// LS Electric XG5000 project: Packing_Machine_NEW1
// PLC NewPLC
// module base 0 slot 0: Input/Output Module:XBC-DN/DP32U (DC 24V Input 16 Contacts, Transistor Output 16 Contacts)
// module base 0 slot 1: Internal Positioning:XBF-PD04E (Position Control  Pulse(LD), Output Type(4 axis))

PROGRAM Program (task: Scan Program)

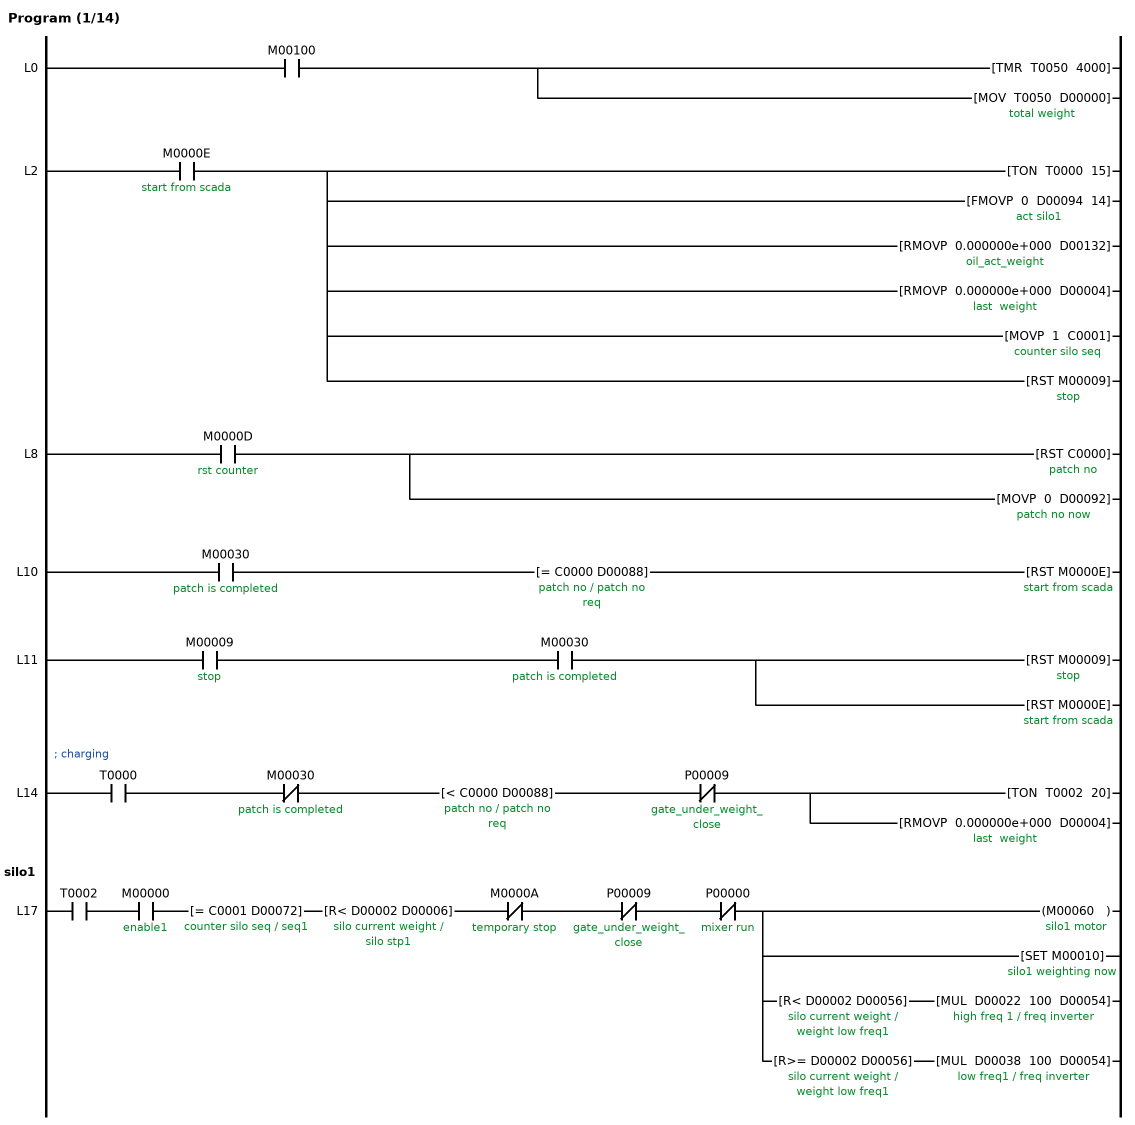
; L0
LOAD      M00100
TMR       T0050 4000
MOV       T0050 D00000	// total weight
; L2
LOAD      M0000E	// start from scada
TON       T0000 15
FMOVP     0 D00094 14	// act silo1
RMOVP     0.000000e+000 D00132	// oil_act_weight
RMOVP     0.000000e+000 D00004	// last  weight
MOVP      1 C0001	// counter silo seq
RST       M00009	// stop
; L8
LOAD      M0000D	// rst counter
RST       C0000	// patch no
MOVP      0 D00092	// patch no now
; L10
LOAD      M00030	// patch is completed
AND=      C0000 D00088	// patch no / patch no req
RST       M0000E	// start from scada
; L11
LOAD      M00009	// stop
AND       M00030	// patch is completed
RST       M00009	// stop
RST       M0000E	// start from scada
// charging
; L14
LOAD      T0000
AND NOT   M00030	// patch is completed
AND<      C0000 D00088	// patch no / patch no req
AND NOT   P00009	// gate_under_weight_close
TON       T0002 20
RMOVP     0.000000e+000 D00004	// last  weight
silo1:
; L17
LOAD      T0002
AND       M00000	// enable1
AND=      C0001 D00072	// counter silo seq / seq1
ANDR<     D00002 D00006	// silo current weight / silo stp1
AND NOT   M0000A	// temporary stop
AND NOT   P00009	// gate_under_weight_close
AND NOT   P00000	// mixer run
OUT       M00060	// silo1 motor
SET       M00010	// silo1 weighting now
MPUSH
ANDR<     D00002 D00056	// silo current weight / weight low freq1
MUL       D00022 100 D00054	// high freq 1 / freq inverter
MPOP
ANDR>=    D00002 D00056	// silo current weight / weight low freq1
MUL       D00038 100 D00054	// low freq1 / freq inverter

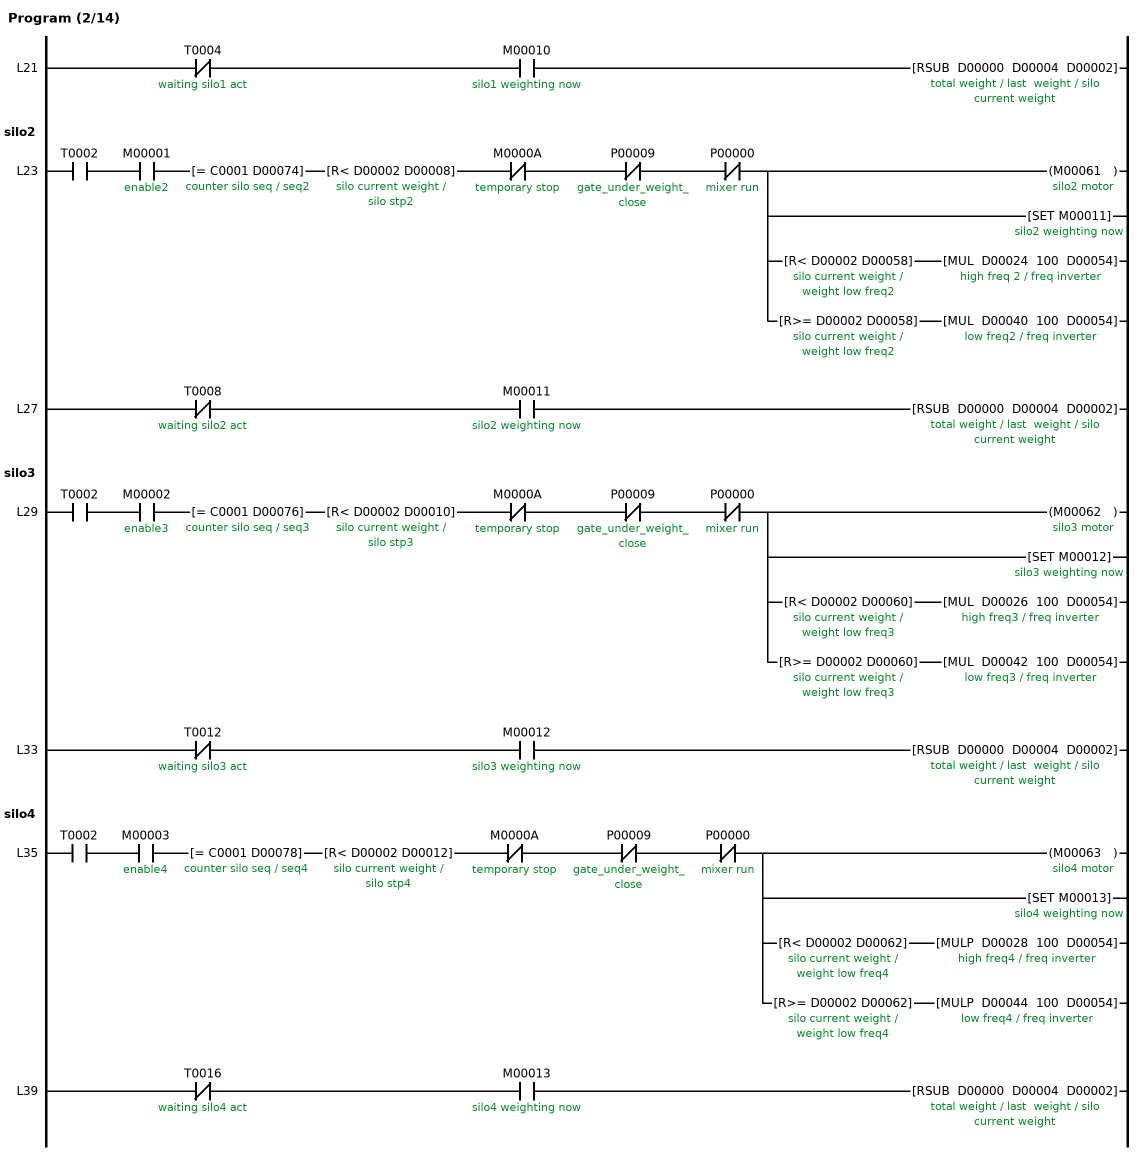
; L21
LOAD NOT  T0004	// waiting silo1 act
AND       M00010	// silo1 weighting now
RSUB      D00000 D00004 D00002	// total weight / last  weight / silo current weight
silo2:
; L23
LOAD      T0002
AND       M00001	// enable2
AND=      C0001 D00074	// counter silo seq / seq2
ANDR<     D00002 D00008	// silo current weight / silo stp2
AND NOT   M0000A	// temporary stop
AND NOT   P00009	// gate_under_weight_close
AND NOT   P00000	// mixer run
OUT       M00061	// silo2 motor
SET       M00011	// silo2 weighting now
MPUSH
ANDR<     D00002 D00058	// silo current weight / weight low freq2
MUL       D00024 100 D00054	// high freq 2 / freq inverter
MPOP
ANDR>=    D00002 D00058	// silo current weight / weight low freq2
MUL       D00040 100 D00054	// low freq2 / freq inverter
; L27
LOAD NOT  T0008	// waiting silo2 act
AND       M00011	// silo2 weighting now
RSUB      D00000 D00004 D00002	// total weight / last  weight / silo current weight
silo3:
; L29
LOAD      T0002
AND       M00002	// enable3
AND=      C0001 D00076	// counter silo seq / seq3
ANDR<     D00002 D00010	// silo current weight / silo stp3
AND NOT   M0000A	// temporary stop
AND NOT   P00009	// gate_under_weight_close
AND NOT   P00000	// mixer run
OUT       M00062	// silo3 motor
SET       M00012	// silo3 weighting now
MPUSH
ANDR<     D00002 D00060	// silo current weight / weight low freq3
MUL       D00026 100 D00054	// high freq3 / freq inverter
MPOP
ANDR>=    D00002 D00060	// silo current weight / weight low freq3
MUL       D00042 100 D00054	// low freq3 / freq inverter
; L33
LOAD NOT  T0012	// waiting silo3 act
AND       M00012	// silo3 weighting now
RSUB      D00000 D00004 D00002	// total weight / last  weight / silo current weight
silo4:
; L35
LOAD      T0002
AND       M00003	// enable4
AND=      C0001 D00078	// counter silo seq / seq4
ANDR<     D00002 D00012	// silo current weight / silo stp4
AND NOT   M0000A	// temporary stop
AND NOT   P00009	// gate_under_weight_close
AND NOT   P00000	// mixer run
OUT       M00063	// silo4 motor
SET       M00013	// silo4 weighting now
MPUSH
ANDR<     D00002 D00062	// silo current weight / weight low freq4
MULP      D00028 100 D00054	// high freq4 / freq inverter
MPOP
ANDR>=    D00002 D00062	// silo current weight / weight low freq4
MULP      D00044 100 D00054	// low freq4 / freq inverter
; L39
LOAD NOT  T0016	// waiting silo4 act
AND       M00013	// silo4 weighting now
RSUB      D00000 D00004 D00002	// total weight / last  weight / silo current weight

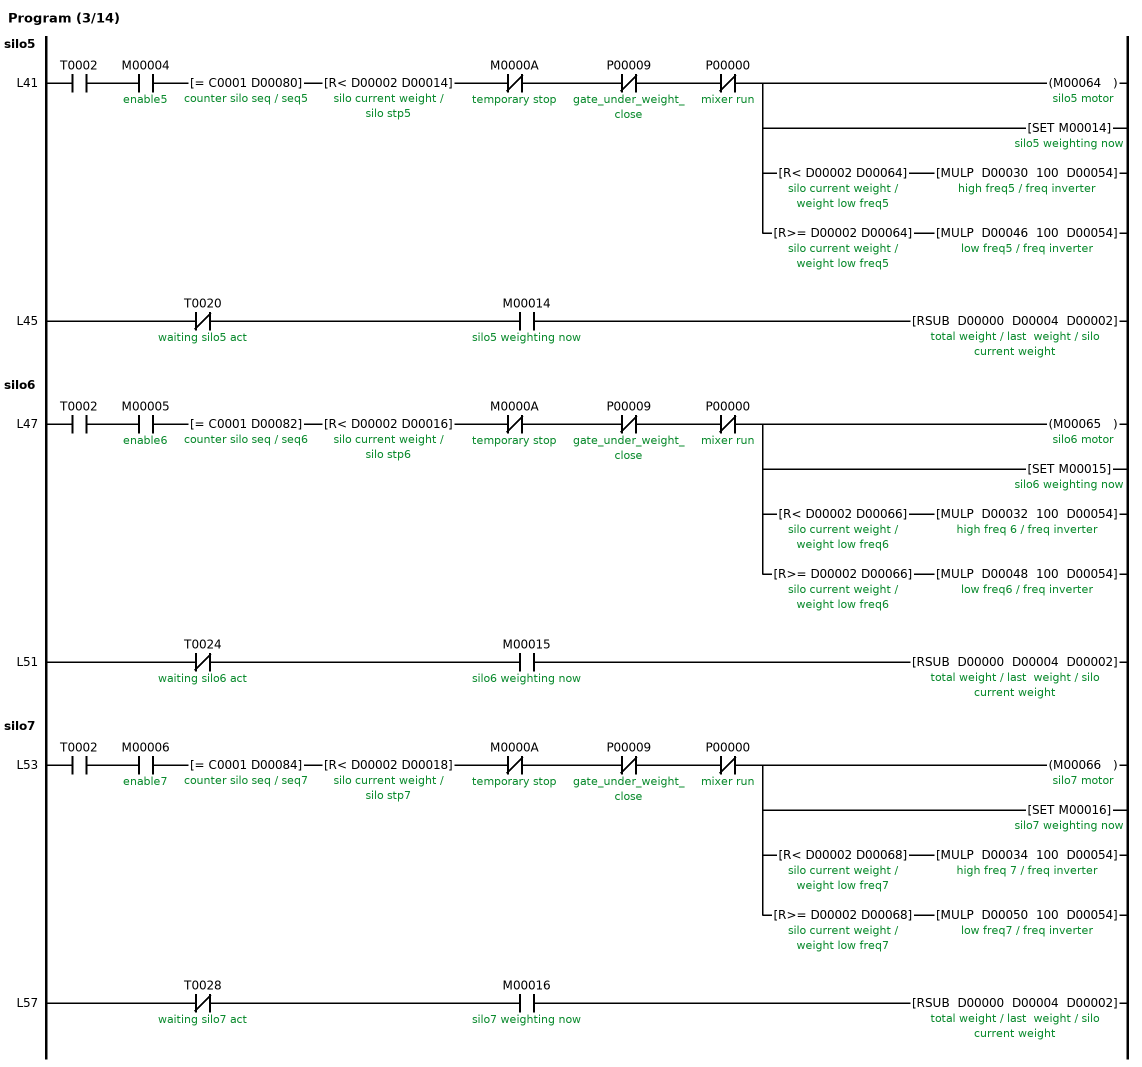
silo5:
; L41
LOAD      T0002
AND       M00004	// enable5
AND=      C0001 D00080	// counter silo seq / seq5
ANDR<     D00002 D00014	// silo current weight / silo stp5
AND NOT   M0000A	// temporary stop
AND NOT   P00009	// gate_under_weight_close
AND NOT   P00000	// mixer run
OUT       M00064	// silo5 motor
SET       M00014	// silo5 weighting now
MPUSH
ANDR<     D00002 D00064	// silo current weight / weight low freq5
MULP      D00030 100 D00054	// high freq5 / freq inverter
MPOP
ANDR>=    D00002 D00064	// silo current weight / weight low freq5
MULP      D00046 100 D00054	// low freq5 / freq inverter
; L45
LOAD NOT  T0020	// waiting silo5 act
AND       M00014	// silo5 weighting now
RSUB      D00000 D00004 D00002	// total weight / last  weight / silo current weight
silo6:
; L47
LOAD      T0002
AND       M00005	// enable6
AND=      C0001 D00082	// counter silo seq / seq6
ANDR<     D00002 D00016	// silo current weight / silo stp6
AND NOT   M0000A	// temporary stop
AND NOT   P00009	// gate_under_weight_close
AND NOT   P00000	// mixer run
OUT       M00065	// silo6 motor
SET       M00015	// silo6 weighting now
MPUSH
ANDR<     D00002 D00066	// silo current weight / weight low freq6
MULP      D00032 100 D00054	// high freq 6 / freq inverter
MPOP
ANDR>=    D00002 D00066	// silo current weight / weight low freq6
MULP      D00048 100 D00054	// low freq6 / freq inverter
; L51
LOAD NOT  T0024	// waiting silo6 act
AND       M00015	// silo6 weighting now
RSUB      D00000 D00004 D00002	// total weight / last  weight / silo current weight
silo7:
; L53
LOAD      T0002
AND       M00006	// enable7
AND=      C0001 D00084	// counter silo seq / seq7
ANDR<     D00002 D00018	// silo current weight / silo stp7
AND NOT   M0000A	// temporary stop
AND NOT   P00009	// gate_under_weight_close
AND NOT   P00000	// mixer run
OUT       M00066	// silo7 motor
SET       M00016	// silo7 weighting now
MPUSH
ANDR<     D00002 D00068	// silo current weight / weight low freq7
MULP      D00034 100 D00054	// high freq 7 / freq inverter
MPOP
ANDR>=    D00002 D00068	// silo current weight / weight low freq7
MULP      D00050 100 D00054	// low freq7 / freq inverter
; L57
LOAD NOT  T0028	// waiting silo7 act
AND       M00016	// silo7 weighting now
RSUB      D00000 D00004 D00002	// total weight / last  weight / silo current weight

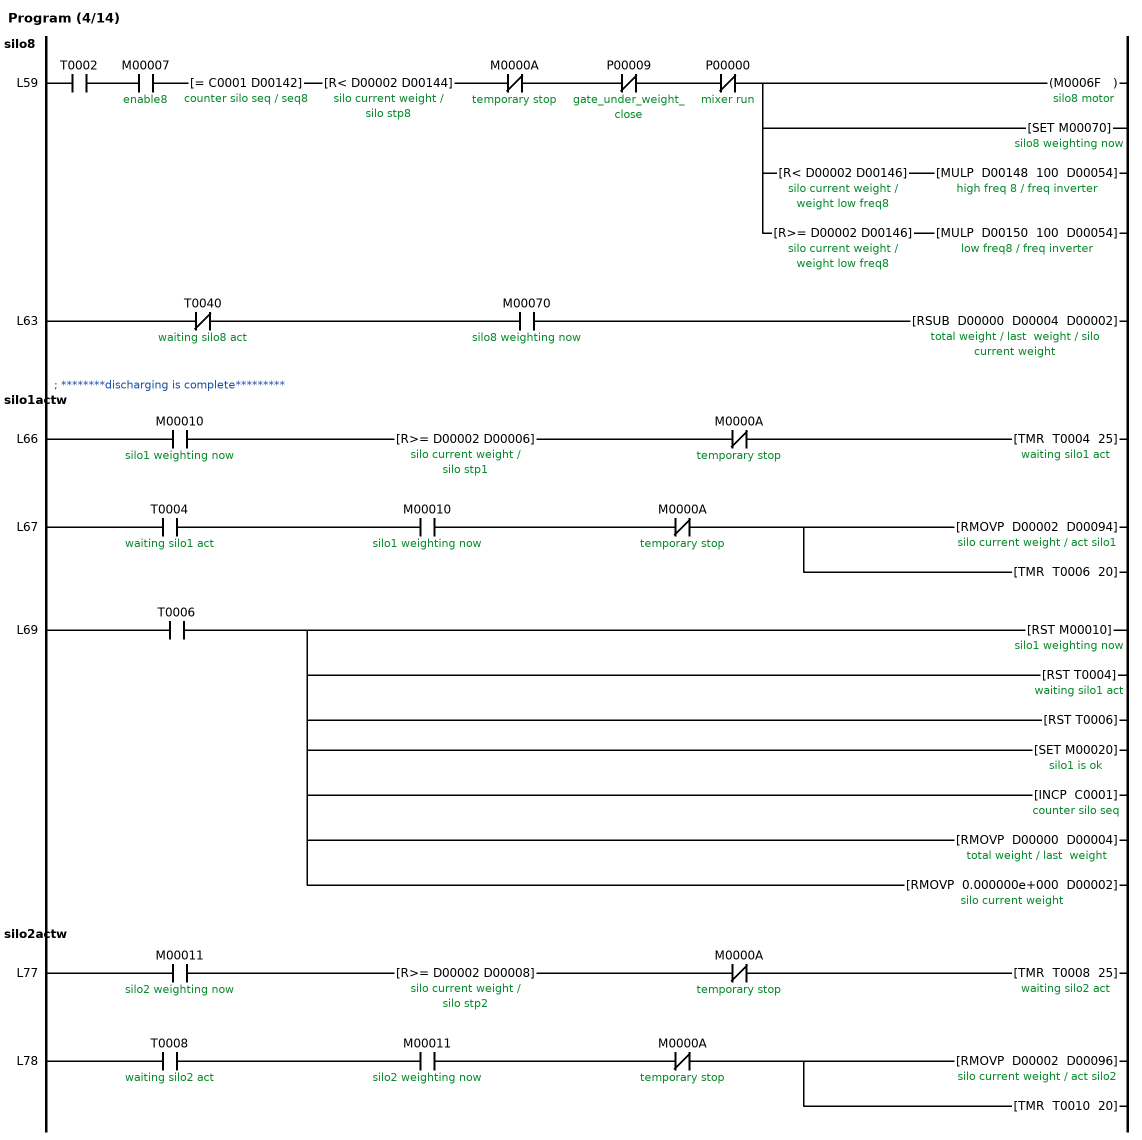
silo8:
; L59
LOAD      T0002
AND       M00007	// enable8
AND=      C0001 D00142	// counter silo seq / seq8
ANDR<     D00002 D00144	// silo current weight / silo stp8
AND NOT   M0000A	// temporary stop
AND NOT   P00009	// gate_under_weight_close
AND NOT   P00000	// mixer run
OUT       M0006F	// silo8 motor
SET       M00070	// silo8 weighting now
MPUSH
ANDR<     D00002 D00146	// silo current weight / weight low freq8
MULP      D00148 100 D00054	// high freq 8 / freq inverter
MPOP
ANDR>=    D00002 D00146	// silo current weight / weight low freq8
MULP      D00150 100 D00054	// low freq8 / freq inverter
; L63
LOAD NOT  T0040	// waiting silo8 act
AND       M00070	// silo8 weighting now
RSUB      D00000 D00004 D00002	// total weight / last  weight / silo current weight
// ********discharging is complete*********
silo1actw:
; L66
LOAD      M00010	// silo1 weighting now
ANDR>=    D00002 D00006	// silo current weight / silo stp1
AND NOT   M0000A	// temporary stop
TMR       T0004 25	// waiting silo1 act
; L67
LOAD      T0004	// waiting silo1 act
AND       M00010	// silo1 weighting now
AND NOT   M0000A	// temporary stop
RMOVP     D00002 D00094	// silo current weight / act silo1
TMR       T0006 20
; L69
LOAD      T0006
RST       M00010	// silo1 weighting now
RST       T0004	// waiting silo1 act
RST       T0006
SET       M00020	// silo1 is ok
INCP      C0001	// counter silo seq
RMOVP     D00000 D00004	// total weight / last  weight
RMOVP     0.000000e+000 D00002	// silo current weight
silo2actw:
; L77
LOAD      M00011	// silo2 weighting now
ANDR>=    D00002 D00008	// silo current weight / silo stp2
AND NOT   M0000A	// temporary stop
TMR       T0008 25	// waiting silo2 act
; L78
LOAD      T0008	// waiting silo2 act
AND       M00011	// silo2 weighting now
AND NOT   M0000A	// temporary stop
RMOVP     D00002 D00096	// silo current weight / act silo2
TMR       T0010 20

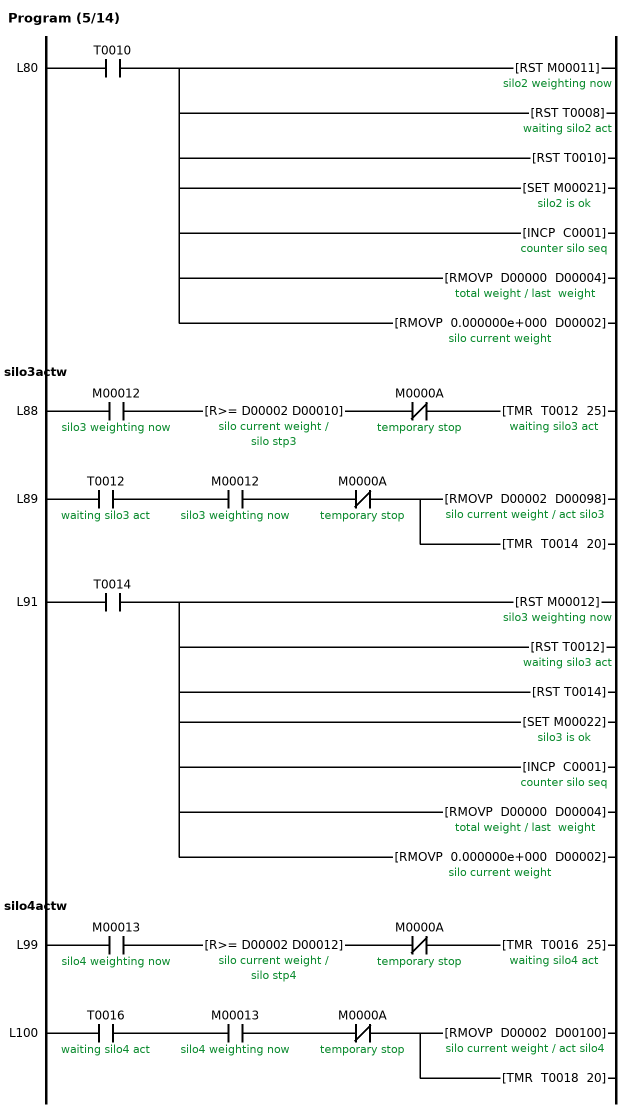
; L80
LOAD      T0010
RST       M00011	// silo2 weighting now
RST       T0008	// waiting silo2 act
RST       T0010
SET       M00021	// silo2 is ok
INCP      C0001	// counter silo seq
RMOVP     D00000 D00004	// total weight / last  weight
RMOVP     0.000000e+000 D00002	// silo current weight
silo3actw:
; L88
LOAD      M00012	// silo3 weighting now
ANDR>=    D00002 D00010	// silo current weight / silo stp3
AND NOT   M0000A	// temporary stop
TMR       T0012 25	// waiting silo3 act
; L89
LOAD      T0012	// waiting silo3 act
AND       M00012	// silo3 weighting now
AND NOT   M0000A	// temporary stop
RMOVP     D00002 D00098	// silo current weight / act silo3
TMR       T0014 20
; L91
LOAD      T0014
RST       M00012	// silo3 weighting now
RST       T0012	// waiting silo3 act
RST       T0014
SET       M00022	// silo3 is ok
INCP      C0001	// counter silo seq
RMOVP     D00000 D00004	// total weight / last  weight
RMOVP     0.000000e+000 D00002	// silo current weight
silo4actw:
; L99
LOAD      M00013	// silo4 weighting now
ANDR>=    D00002 D00012	// silo current weight / silo stp4
AND NOT   M0000A	// temporary stop
TMR       T0016 25	// waiting silo4 act
; L100
LOAD      T0016	// waiting silo4 act
AND       M00013	// silo4 weighting now
AND NOT   M0000A	// temporary stop
RMOVP     D00002 D00100	// silo current weight / act silo4
TMR       T0018 20

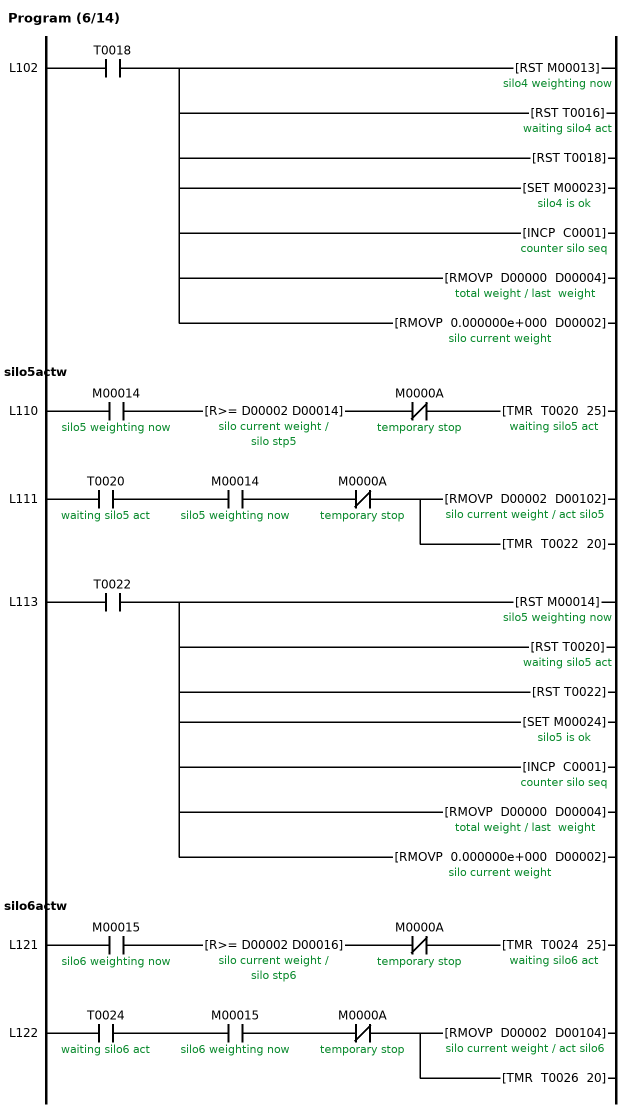
; L102
LOAD      T0018
RST       M00013	// silo4 weighting now
RST       T0016	// waiting silo4 act
RST       T0018
SET       M00023	// silo4 is ok
INCP      C0001	// counter silo seq
RMOVP     D00000 D00004	// total weight / last  weight
RMOVP     0.000000e+000 D00002	// silo current weight
silo5actw:
; L110
LOAD      M00014	// silo5 weighting now
ANDR>=    D00002 D00014	// silo current weight / silo stp5
AND NOT   M0000A	// temporary stop
TMR       T0020 25	// waiting silo5 act
; L111
LOAD      T0020	// waiting silo5 act
AND       M00014	// silo5 weighting now
AND NOT   M0000A	// temporary stop
RMOVP     D00002 D00102	// silo current weight / act silo5
TMR       T0022 20
; L113
LOAD      T0022
RST       M00014	// silo5 weighting now
RST       T0020	// waiting silo5 act
RST       T0022
SET       M00024	// silo5 is ok
INCP      C0001	// counter silo seq
RMOVP     D00000 D00004	// total weight / last  weight
RMOVP     0.000000e+000 D00002	// silo current weight
silo6actw:
; L121
LOAD      M00015	// silo6 weighting now
ANDR>=    D00002 D00016	// silo current weight / silo stp6
AND NOT   M0000A	// temporary stop
TMR       T0024 25	// waiting silo6 act
; L122
LOAD      T0024	// waiting silo6 act
AND       M00015	// silo6 weighting now
AND NOT   M0000A	// temporary stop
RMOVP     D00002 D00104	// silo current weight / act silo6
TMR       T0026 20

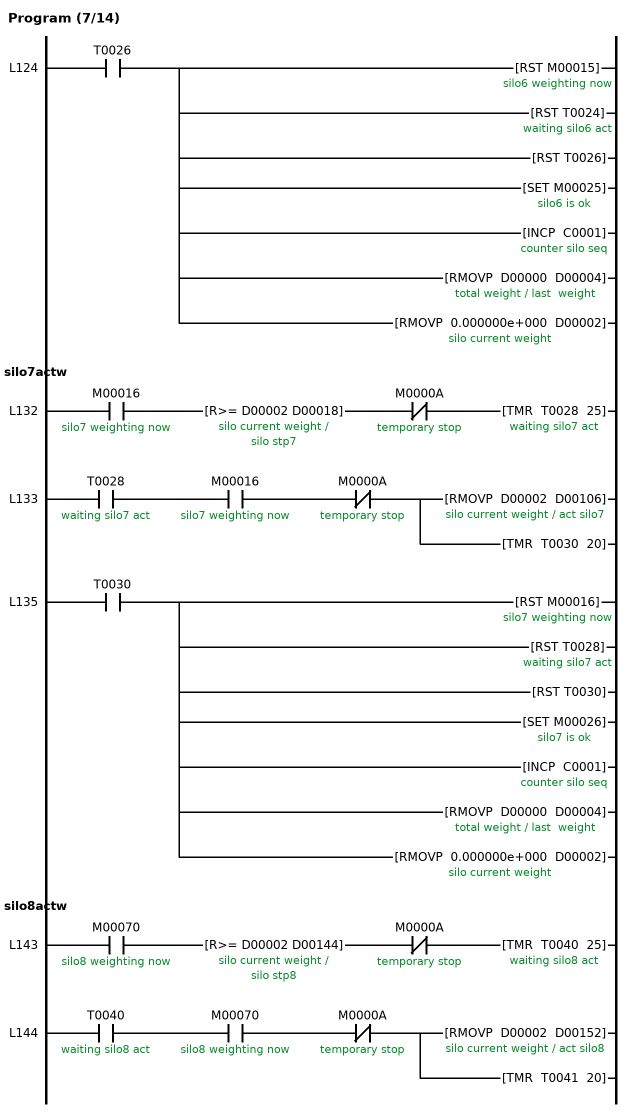
; L124
LOAD      T0026
RST       M00015	// silo6 weighting now
RST       T0024	// waiting silo6 act
RST       T0026
SET       M00025	// silo6 is ok
INCP      C0001	// counter silo seq
RMOVP     D00000 D00004	// total weight / last  weight
RMOVP     0.000000e+000 D00002	// silo current weight
silo7actw:
; L132
LOAD      M00016	// silo7 weighting now
ANDR>=    D00002 D00018	// silo current weight / silo stp7
AND NOT   M0000A	// temporary stop
TMR       T0028 25	// waiting silo7 act
; L133
LOAD      T0028	// waiting silo7 act
AND       M00016	// silo7 weighting now
AND NOT   M0000A	// temporary stop
RMOVP     D00002 D00106	// silo current weight / act silo7
TMR       T0030 20
; L135
LOAD      T0030
RST       M00016	// silo7 weighting now
RST       T0028	// waiting silo7 act
RST       T0030
SET       M00026	// silo7 is ok
INCP      C0001	// counter silo seq
RMOVP     D00000 D00004	// total weight / last  weight
RMOVP     0.000000e+000 D00002	// silo current weight
silo8actw:
; L143
LOAD      M00070	// silo8 weighting now
ANDR>=    D00002 D00144	// silo current weight / silo stp8
AND NOT   M0000A	// temporary stop
TMR       T0040 25	// waiting silo8 act
; L144
LOAD      T0040	// waiting silo8 act
AND       M00070	// silo8 weighting now
AND NOT   M0000A	// temporary stop
RMOVP     D00002 D00152	// silo current weight / act silo8
TMR       T0041 20

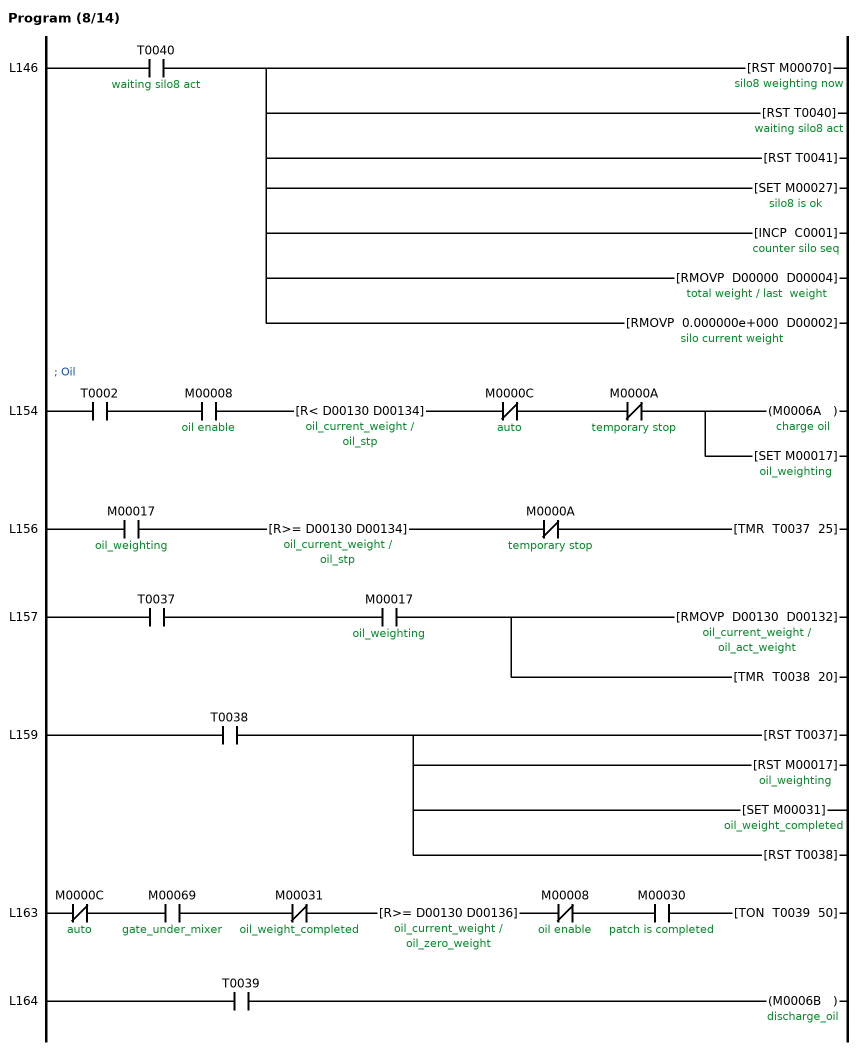
; L146
LOAD      T0040	// waiting silo8 act
RST       M00070	// silo8 weighting now
RST       T0040	// waiting silo8 act
RST       T0041
SET       M00027	// silo8 is ok
INCP      C0001	// counter silo seq
RMOVP     D00000 D00004	// total weight / last  weight
RMOVP     0.000000e+000 D00002	// silo current weight
// Oil
; L154
LOAD      T0002
AND       M00008	// oil enable
ANDR<     D00130 D00134	// oil_current_weight / oil_stp
AND NOT   M0000C	// auto
AND NOT   M0000A	// temporary stop
OUT       M0006A	// charge oil
SET       M00017	// oil_weighting
; L156
LOAD      M00017	// oil_weighting
ANDR>=    D00130 D00134	// oil_current_weight / oil_stp
AND NOT   M0000A	// temporary stop
TMR       T0037 25
; L157
LOAD      T0037
AND       M00017	// oil_weighting
RMOVP     D00130 D00132	// oil_current_weight / oil_act_weight
TMR       T0038 20
; L159
LOAD      T0038
RST       T0037
RST       M00017	// oil_weighting
SET       M00031	// oil_weight_completed
RST       T0038
; L163
LOAD NOT  M0000C	// auto
AND       M00069	// gate_under_mixer
AND NOT   M00031	// oil_weight_completed
ANDR>=    D00130 D00136	// oil_current_weight / oil_zero_weight
AND NOT   M00008	// oil enable
AND       M00030	// patch is completed
TON       T0039 50
; L164
LOAD      T0039
OUT       M0006B	// discharge_oil

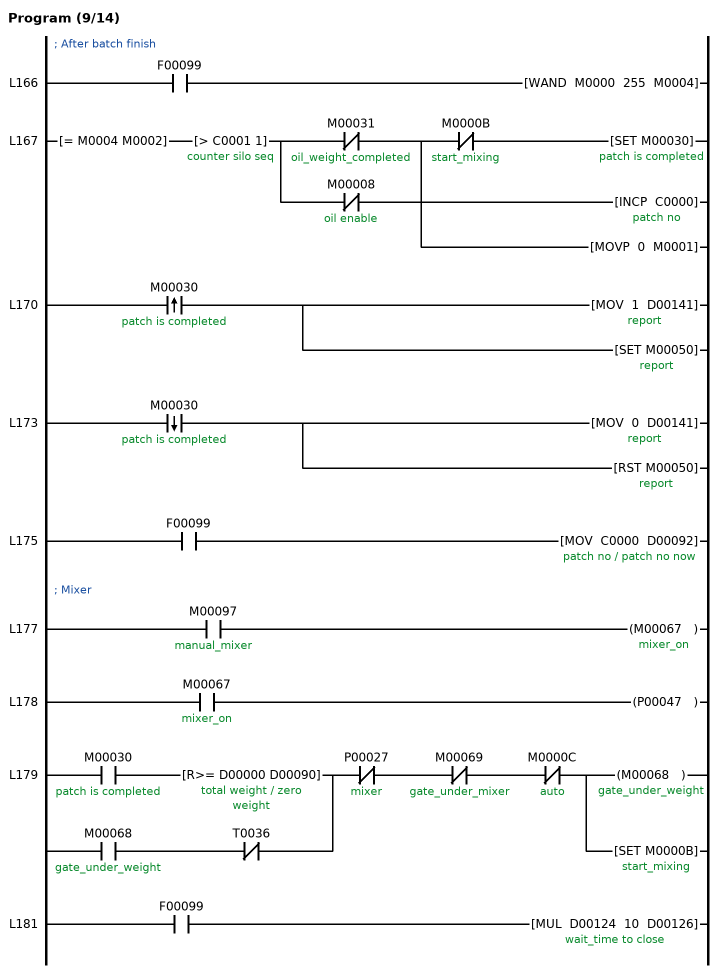
// After batch finish
; L166
LOAD      F00099
WAND      M0000 255 M0004
; L167
LOAD=     M0004 M0002
AND>      C0001 1	// counter silo seq
LOAD NOT  M00031	// oil_weight_completed
OR NOT    M00008	// oil enable
AND LOAD
MPUSH
AND NOT   M0000B	// start_mixing
SET       M00030	// patch is completed
MPOP
INCP      C0000	// patch no
MOVP      0 M0001
; L170
LOADP     M00030	// patch is completed
MOV       1 D00141	// report
SET       M00050	// report
; L173
LOADN     M00030	// patch is completed
MOV       0 D00141	// report
RST       M00050	// report
; L175
LOAD      F00099
MOV       C0000 D00092	// patch no / patch no now
// Mixer
; L177
LOAD      M00097	// manual_mixer
OUT       M00067	// mixer_on
; L178
LOAD      M00067	// mixer_on
OUT       P00047
; L179
LOAD      M00030	// patch is completed
ANDR>=    D00000 D00090	// total weight / zero weight
LOAD      M00068	// gate_under_weight
AND NOT   T0036
OR LOAD
AND NOT   P00027	// mixer
AND NOT   M00069	// gate_under_mixer
AND NOT   M0000C	// auto
OUT       M00068	// gate_under_weight
SET       M0000B	// start_mixing
; L181
LOAD      F00099
MUL       D00124 10 D00126	// wait_time to close

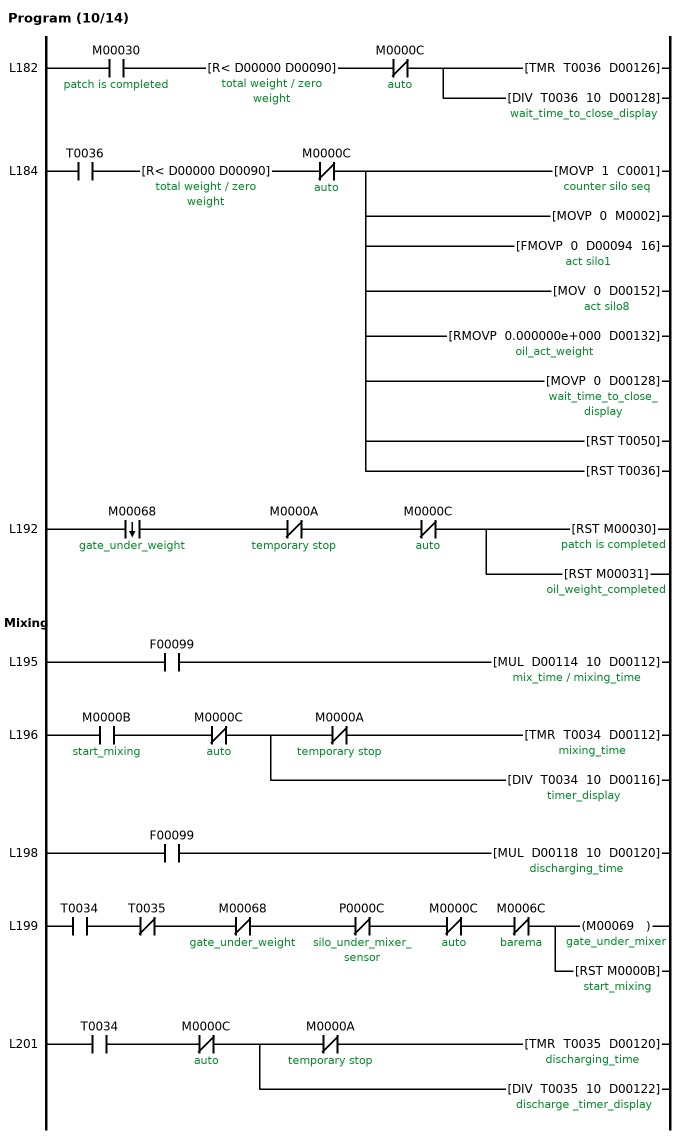
; L182
LOAD      M00030	// patch is completed
ANDR<     D00000 D00090	// total weight / zero weight
AND NOT   M0000C	// auto
TMR       T0036 D00126
DIV       T0036 10 D00128	// wait_time_to_close_display
; L184
LOAD      T0036
ANDR<     D00000 D00090	// total weight / zero weight
AND NOT   M0000C	// auto
MOVP      1 C0001	// counter silo seq
MOVP      0 M0002
FMOVP     0 D00094 16	// act silo1
MOV       0 D00152	// act silo8
RMOVP     0.000000e+000 D00132	// oil_act_weight
MOVP      0 D00128	// wait_time_to_close_display
RST       T0050
RST       T0036
; L192
LOADN     M00068	// gate_under_weight
AND NOT   M0000A	// temporary stop
AND NOT   M0000C	// auto
RST       M00030	// patch is completed
RST       M00031	// oil_weight_completed
Mixing:
; L195
LOAD      F00099
MUL       D00114 10 D00112	// mix_time / mixing_time
; L196
LOAD      M0000B	// start_mixing
AND NOT   M0000C	// auto
MPUSH
AND NOT   M0000A	// temporary stop
TMR       T0034 D00112	// mixing_time
MPOP
DIV       T0034 10 D00116	// timer_display
; L198
LOAD      F00099
MUL       D00118 10 D00120	// discharging_time
; L199
LOAD      T0034
AND NOT   T0035
AND NOT   M00068	// gate_under_weight
AND NOT   P0000C	// silo_under_mixer_sensor
AND NOT   M0000C	// auto
AND NOT   M0006C	// barema
OUT       M00069	// gate_under_mixer
RST       M0000B	// start_mixing
; L201
LOAD      T0034
AND NOT   M0000C	// auto
MPUSH
AND NOT   M0000A	// temporary stop
TMR       T0035 D00120	// discharging_time
MPOP
DIV       T0035 10 D00122	// discharge _timer_display

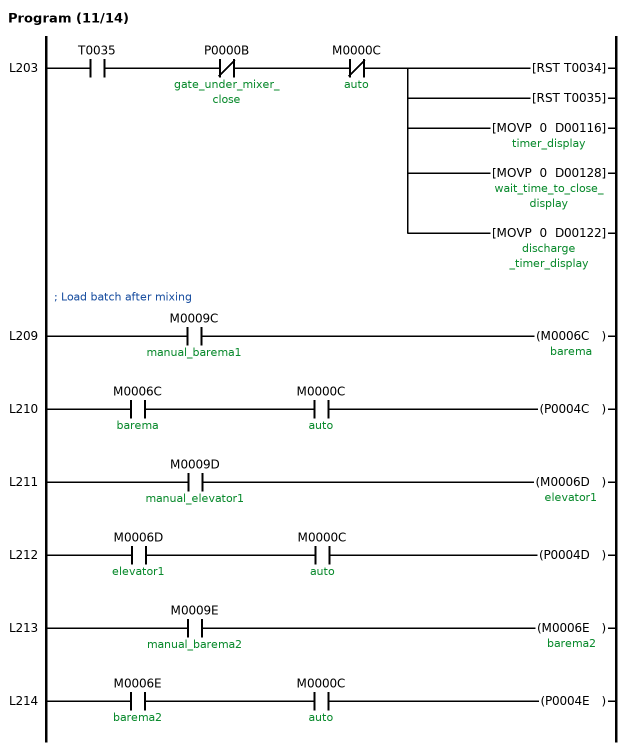
; L203
LOAD      T0035
AND NOT   P0000B	// gate_under_mixer_close
AND NOT   M0000C	// auto
RST       T0034
RST       T0035
MOVP      0 D00116	// timer_display
MOVP      0 D00128	// wait_time_to_close_display
MOVP      0 D00122	// discharge _timer_display
// Load batch after mixing
; L209
LOAD      M0009C	// manual_barema1
OUT       M0006C	// barema
; L210
LOAD      M0006C	// barema
AND       M0000C	// auto
OUT       P0004C
; L211
LOAD      M0009D	// manual_elevator1
OUT       M0006D	// elevator1
; L212
LOAD      M0006D	// elevator1
AND       M0000C	// auto
OUT       P0004D
; L213
LOAD      M0009E	// manual_barema2
OUT       M0006E	// barema2
; L214
LOAD      M0006E	// barema2
AND       M0000C	// auto
OUT       P0004E

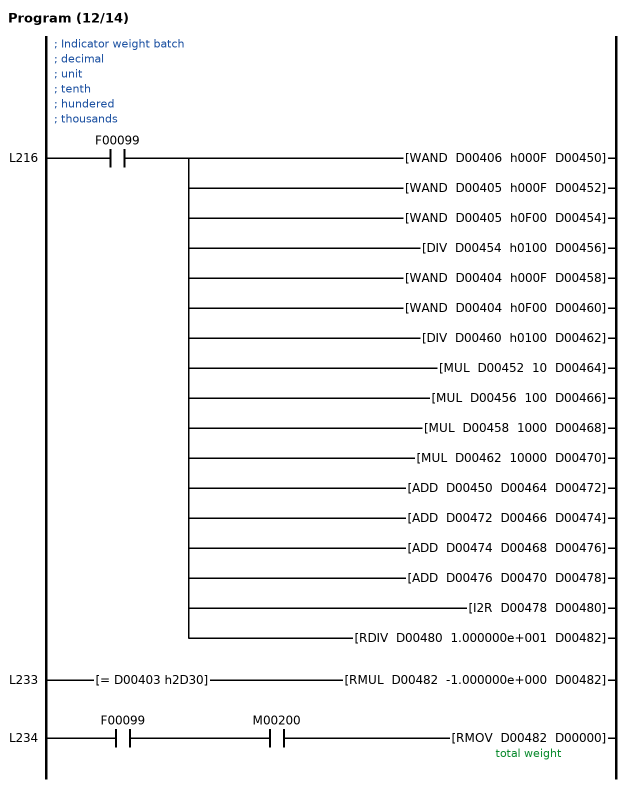
// Indicator weight batch
; L216
LOAD      F00099
WAND      D00406 h000F D00450
WAND      D00405 h000F D00452
WAND      D00405 h0F00 D00454
DIV       D00454 h0100 D00456
WAND      D00404 h000F D00458
WAND      D00404 h0F00 D00460
DIV       D00460 h0100 D00462
MUL       D00452 10 D00464
MUL       D00456 100 D00466
MUL       D00458 1000 D00468
MUL       D00462 10000 D00470
ADD       D00450 D00464 D00472
ADD       D00472 D00466 D00474
ADD       D00474 D00468 D00476
ADD       D00476 D00470 D00478
I2R       D00478 D00480
RDIV      D00480 1.000000e+001 D00482
// output comment: decimal
// output comment: unit
// output comment: tenth
// output comment: hundered
// output comment: thousands
; L233
LOAD=     D00403 h2D30
RMUL      D00482 -1.000000e+000 D00482
; L234
LOAD      F00099
AND       M00200
RMOV      D00482 D00000	// total weight

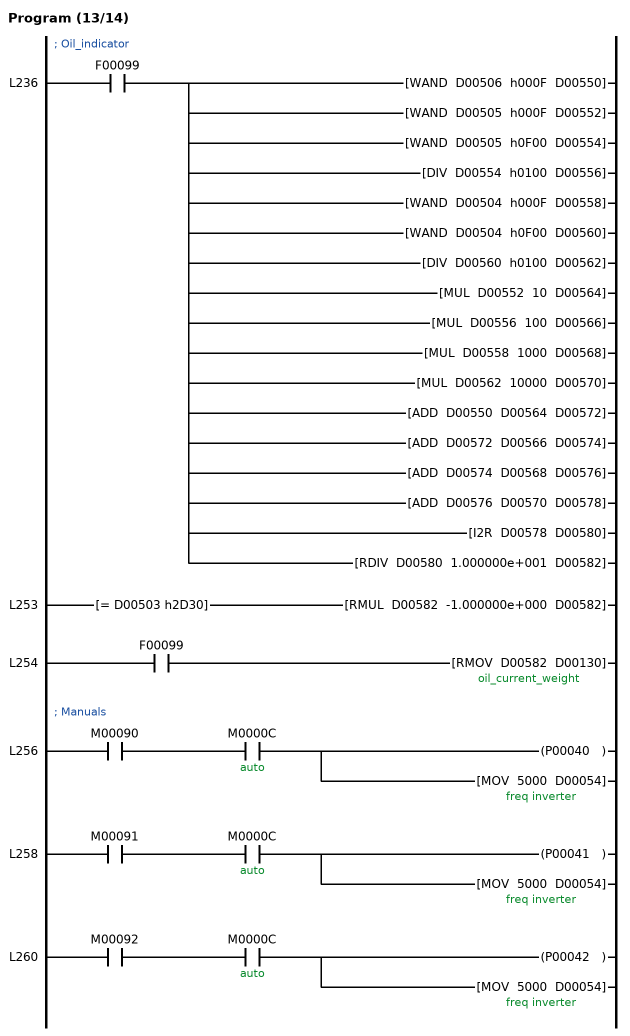
// Oil_indicator
; L236
LOAD      F00099
WAND      D00506 h000F D00550
WAND      D00505 h000F D00552
WAND      D00505 h0F00 D00554
DIV       D00554 h0100 D00556
WAND      D00504 h000F D00558
WAND      D00504 h0F00 D00560
DIV       D00560 h0100 D00562
MUL       D00552 10 D00564
MUL       D00556 100 D00566
MUL       D00558 1000 D00568
MUL       D00562 10000 D00570
ADD       D00550 D00564 D00572
ADD       D00572 D00566 D00574
ADD       D00574 D00568 D00576
ADD       D00576 D00570 D00578
I2R       D00578 D00580
RDIV      D00580 1.000000e+001 D00582
; L253
LOAD=     D00503 h2D30
RMUL      D00582 -1.000000e+000 D00582
; L254
LOAD      F00099
RMOV      D00582 D00130	// oil_current_weight
// Manuals
; L256
LOAD      M00090
AND       M0000C	// auto
OUT       P00040
MOV       5000 D00054	// freq inverter
; L258
LOAD      M00091
AND       M0000C	// auto
OUT       P00041
MOV       5000 D00054	// freq inverter
; L260
LOAD      M00092
AND       M0000C	// auto
OUT       P00042
MOV       5000 D00054	// freq inverter

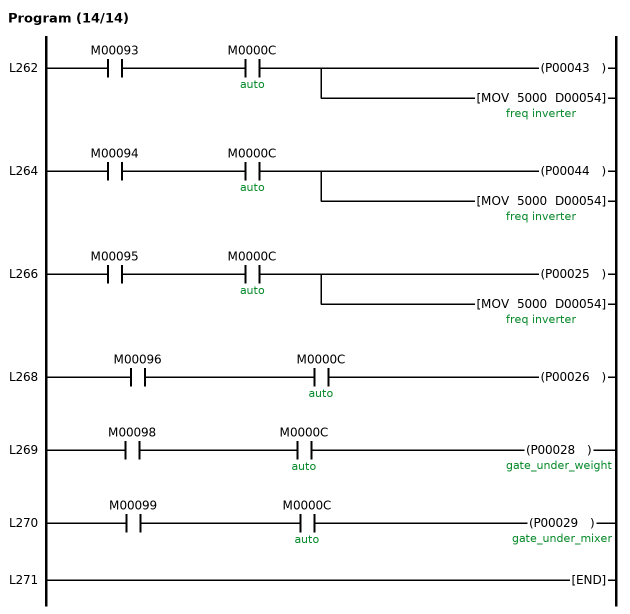
; L262
LOAD      M00093
AND       M0000C	// auto
OUT       P00043
MOV       5000 D00054	// freq inverter
; L264
LOAD      M00094
AND       M0000C	// auto
OUT       P00044
MOV       5000 D00054	// freq inverter
; L266
LOAD      M00095
AND       M0000C	// auto
OUT       P00025
MOV       5000 D00054	// freq inverter
; L268
LOAD      M00096
AND       M0000C	// auto
OUT       P00026
; L269
LOAD      M00098
AND       M0000C	// auto
OUT       P00028	// gate_under_weight
; L270
LOAD      M00099
AND       M0000C	// auto
OUT       P00029	// gate_under_mixer
; L271
END

PROGRAM inverter&outputs&inputs (task: Scan Program)

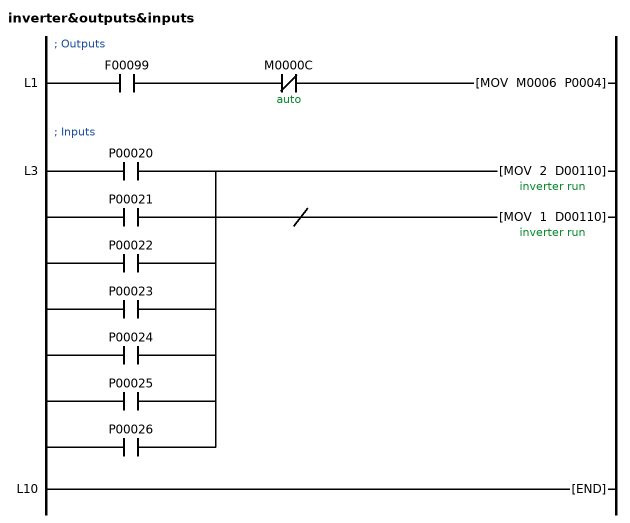
// Outputs
; L1
LOAD      F00099
AND NOT   M0000C	// auto
MOV       M0006 P0004
// Inputs
; L3
LOAD      P00020
OR        P00021
OR        P00022
OR        P00023
OR        P00024
OR        P00025
OR        P00026
MOV       2 D00110	// inverter run
NOT
MOV       1 D00110	// inverter run
; L10
END

VARIABLES AND COMMENTS (devices not used above)
D00020	WORD	silo stp 8
D00036	WORD	high freq 8
D00052	WORD	low freq8
D00070	WORD	weight low freq8
D00086	WORD	seq8
D00108	WORD	act silo8
P00008	BIT	gate_under_weight_open
P0000A	BIT	gate_under_mixer_open
P0002A	BIT	barema2
P0002D	BIT	elevator1
P0002E	BIT	barema2
D00140	WORD	oil_stp
P0002C	BIT	barema
M00032	BIT	patch enter